// TIA Portal V19 export
ORGANIZATION_BLOCK "Time error interrupt"   // OB80, STL, TimeErrorInterrupt
{ S7_Optimized_Access := 'FALSE' }
   VAR_TEMP
      EV_CLASS : Byte;   // 16#35: Event class 3, Entering event state, Internal fault event
      FLT_ID : Byte;   // Fault identifier
      PRIORITY : Byte;   // Priority of OB Execution
      OB_NUMBR : Byte;   // OB number
      RESERVED_1 : Byte;   // Reserved for system
      RESERVED_2 : Byte;   // Reserved for system
      ERROR_INFO : Word;   // Error information on event
      ERR_EV_CLASS : Byte;   // Class of event causing the error
      ERR_EV_NUM : Byte;   // Number of event causing the error
      OB_PRIORITY : Byte;   // Priority of OB causing the error
      OB_NUM : Byte;   // Number of OB causing the error
      DATE_TIME : Date_And_Time;   // Date and time OB started
   END_VAR
BEGIN
END_ORGANIZATION_BLOCK
